// TIA Portal V17 export
// export: Created 2024-12-18T10:10:23.0407237Z, ExportSetting WithDefaults, DisplayName Totally Integrated Automation Portal, DisplayVersion V17, DisplayName TIA Portal Openness, DisplayVersion V17, DisplayName TIA Portal Version Control Interface, DisplayVersion V17, DisplayName STEP 7 Professional, DisplayVersion V17, DisplayName STEP 7 Safety, DisplayVersion V17, DisplayName WinCC Advanced / Unified PC, DisplayVersion V17
FUNCTION_BLOCK "Move Average Test"   // FB5, LAD
{ S7_Optimized_Access := 'TRUE' }
VERSION : 0.1
// stored: AutoNumber true, IsIECCheckEnabled false, IsRetainMemResEnabled false, MemoryReserve 100, SetENOAutomatically false, UDAEnableTagReadback false
   VAR_TEMP   // added for the SCL form of the ladder/FBD networks
      _w1 : Bool;
   END_VAR
BEGIN

REGION Network 1
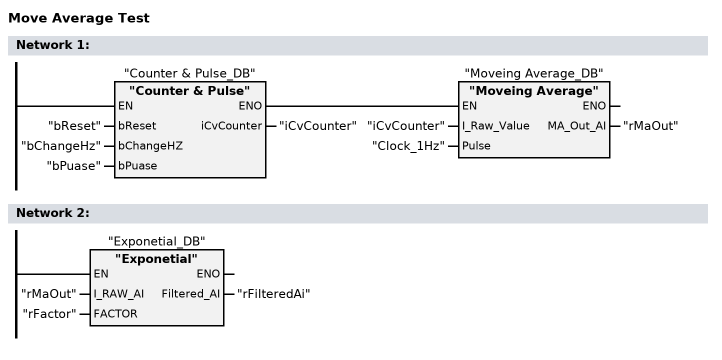
   RUNG wire#powerrail
      "Counter & Pulse_DB"(bReset := "bReset", bChangeHZ := "bChangeHz", bPuase := "bPuase", iCvCounter => "iCvCounter")
      "Moveing Average_DB"(I_Raw_Value := "iCvCounter", Pulse := "Clock_1Hz", MA_Out_AI => "rMaOut")
   END_RUNG
   // the same network as SCL:
   "Counter & Pulse_DB"(bReset := "bReset",   // "Counter & Pulse"
                        bChangeHZ := "bChangeHz",
                        bPuase := "bPuase",
                        iCvCounter => "iCvCounter",
                        ENO => #_w1);
   IF #_w1 THEN
       "Moveing Average_DB"(I_Raw_Value := "iCvCounter", Pulse := "Clock_1Hz", MA_Out_AI => "rMaOut");   // "Moveing Average"
   END_IF;
END_REGION

REGION Network 2
   RUNG wire#powerrail
      "Exponetial_DB"(I_RAW_AI := "rMaOut", FACTOR := "rFactor", Filtered_AI => "rFilteredAi")
   END_RUNG
   // the same network as SCL:
   "Exponetial_DB"(I_RAW_AI := "rMaOut", FACTOR := "rFactor", Filtered_AI => "rFilteredAi");   // "Exponetial"
END_REGION
END_FUNCTION_BLOCK
